// TIA Portal V18 export
FUNCTION "TEMPLATE--v1.1--00_Only for Commissioning" : Void   // FC4, F_LAD
TITLE = bypass activation by profinet node to use during commissioning
{ S7_Optimized_Access := 'TRUE' }
// 1.0 First Emission
// 1.1 Aligned Syntax to signal_types.csv of the py_builder
BEGIN

REGION Network 1: !!NetworkComment$$
   // One network per node
   // TRUE if the node is not ready to be used
   // FALSE if the node is ready
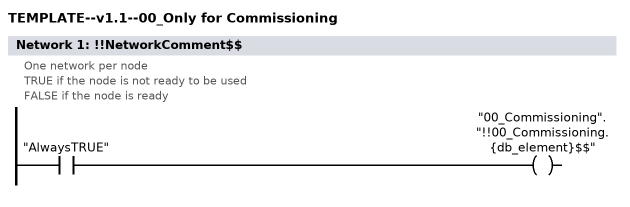
   RUNG wire#powerrail
      Contact( "AlwaysTRUE" )
      Coil( "00_Commissioning"."!!00_Commissioning.{db_element}$$" )
   END_RUNG
   // the same network as SCL:
   "00_Commissioning"."!!00_Commissioning.{db_element}$$" := "AlwaysTRUE";
END_REGION
END_FUNCTION
